{attribute 'enable_dynamic_creation'}	
{attribute 'no_explicit_call' := 'do not call this function block directly'} 
FUNCTION_BLOCK EmptyException EXTENDS Exception
VAR
	_ClassName : STRING := __POUNAME();
END_VAR

{attribute 'monitoring' := 'call'}
PROPERTY ClassName : STRING
GET
ClassName := _ClassName;
END_GET
END_PROPERTY

METHOD Clone : IObject
VAR
	exceptionClone : POINTER TO EmptyException;
END_VAR
exceptionClone := __NEW(EmptyException);

Clone := exceptionClone^;
END_METHOD

{attribute 'monitoring' := 'call'}
PROPERTY Empty : BOOL
GET
Empty := TRUE;
END_GET
END_PROPERTY

METHOD GetMessage : ERROR_MESSAGE
VAR_INPUT
	showTimestamp : BOOL := FALSE;
	showSource : BOOL := FALSE;
END_VAR
GetMessage := "";
END_METHOD

END_FUNCTION_BLOCK

(* stored: Version 1.1.0.1
   POU EmptyException: Id {301384fd-c915-4720-bfde-f90d2dca7ba2}, SpecialFunc None
   Property ClassName: Id {93378995-609b-4770-9943-b61b37cce5dc}
   Get Get: Id {fb4c03aa-4f57-416b-9108-8190d221402d}
   Method Clone: Id {0d6feffe-1bce-43f3-82f4-b46d05cd59ad}
   Property Empty: Id {3252003c-e082-4928-b9ff-3c898a649839}
   Get Get: Id {cbba38a8-2d90-487c-9c38-f866c56d3d30}
   Method GetMessage: Id {33c18aa6-310f-4a0b-a896-a83149c61777} *)
